PROGRAM MAIN
VAR
	Wert_1: INT;
END_VAR

Wert_1:=Wert_1+1;
IF Wert_1>1000 THEN
	Wert_1:=1;
END_IF

END_PROGRAM

(* stored: Version 1.1.0.1, ProductVersion 3.1.4022.3
   POU MAIN: Id {a76eeec2-165b-4d87-90fa-0dbc686344d8}, SpecialFunc None *)
